(* Logix 5000 project; controller BreakGroup_US vendor 1 type 14 code 211 rev 32.16; software revision 32.05 *)

TASK MainTask (continuous, watchdog 500 ms) : MainProgram
TASK MCP_Panel (periodic, rate 50 ms, priority 10, watchdog 500 ms) : Station_10, Station_20, Station_30, Station_40, Station_50, Station_60, Station_70, Station_80, Gantry_01_Vertical, Gantry_01_Horizontal, Gantry_01_Gripper
TASK RCP_Panel (periodic, rate 50 ms, priority 9, watchdog 500 ms) : Gantry_02_Horizontal, Gantry_02_Vertical, Gantry_02_Gripper, Gantry_02_Tilter, Station_90, Oil_Tank_Lift, Station_100, Station_110, Station_120
TASK SafetyTask (periodic, rate 20 ms, priority 10, watchdog 20 ms, safety) : SafetyProgram

MODULES
   Local : vendor 1 type 14 code 211 (ICP 0, rev 32.16)
      POINT_IO : vendor 1 type 12 code 200 (Ethernet 192.168.1.4, ICP 2, rev 11.1)
           MCP_PT01:1:I.0   // Trolley-1 Locking Cylinder Extended
           MCP_PT01:1:I.1   // Trolley-1 Locking Cylinder Retracted
           MCP_PT01:1:I.2   // Trolley Present Sensor
           MCP_PT01:1:I.3   // Trolley Top Side Product Present Sensors
           MCP_PT01:1:I.4   // Trolley-1 Locking Cylinder Extended
           MCP_PT01:1:I.5   // Trolley-1 Locking Cylinder Retracted
           MCP_PT01:1:I.6   // Trolley Present Sensor
         Servo_RCP : vendor 315 type 14 code 24 (Ethernet 192.168.1.12, rev 1.1, StandardDataDriven RPI 20 ms)
         STN_50_INDEX : vendor 315 type 43 code 25 (Ethernet 192.168.1.30, rev 1.1, StandardDataDriven RPI 20 ms)
         Servo_MCP : vendor 315 type 14 code 24 (Ethernet 192.168.1.11, rev 1.1, StandardDataDriven RPI 20 ms)
         STN_100_INDEX : vendor 315 type 43 code 25 (Ethernet 192.168.1.31, rev 1.1, StandardDataDriven RPI 20 ms)
         STN_110_INDEX : vendor 315 type 43 code 25 (Ethernet 192.168.1.32, rev 1.1, StandardDataDriven RPI 20 ms)
         STN_120_INDEX : vendor 315 type 43 code 25 (Ethernet 192.168.1.33, rev 1.1, StandardDataDriven RPI 20 ms)
         MCP_PT01 : 1734-AENTR (Ethernet 192.168.1.7, rev 7.14, Output RPI 20 ms)
             : 1734-IB8 (PointIO 20, rev 3.1)
             : 1734-IB8 (PointIO 8, rev 3.1)
             : 1734-IB8 (PointIO 7, rev 3.1)
            Slot_01 : 1734-IB8 (PointIO 1, rev 3.1)
             : 1734-IB8 (PointIO 5, rev 3.1)
             : 1734-IB8 (PointIO 18, rev 3.1)
             : 1734-IB8 (PointIO 21, rev 3.1)
             : 1734-IB8 (PointIO 9, rev 3.1)
             : 1734-IB8 (PointIO 10, rev 3.1)
             : 1734-IB8 (PointIO 23, rev 3.1)
             : 1734-IB8 (PointIO 2, rev 3.1)
             : 1734-IB8 (PointIO 16, rev 3.1)
             : 1734-IB8 (PointIO 11, rev 3.1)
             : 1734-IB8 (PointIO 17, rev 3.1)
             : 1734-IB8 (PointIO 14, rev 3.1)
             : 1734-IB8 (PointIO 6, rev 3.1)
             : 1734-IB8 (PointIO 24, rev 3.1)
             : 1734-IB8 (PointIO 19, rev 3.1)
             : 1734-IB8 (PointIO 15, rev 3.1)
             : 1734-IB8 (PointIO 22, rev 3.1)
             : 1734-IB8 (PointIO 13, rev 3.1)
             : 1734-IB8 (PointIO 4, rev 3.1)
             : 1734-IB8 (PointIO 12, rev 3.1)
             : 1734-IB8 (PointIO 3, rev 3.1)
             : 1734-OB8 (PointIO 35, rev 3.1)
             : 1734-OB8 (PointIO 30, rev 3.1)
             : 1734-OB8 (PointIO 25, rev 3.1)
             : 1734-OB8 (PointIO 29, rev 3.1)
             : 1734-OB8 (PointIO 34, rev 3.1)
             : 1734-OB8 (PointIO 32, rev 3.1)
             : 1734-OB8 (PointIO 28, rev 3.1)
             : 1734-OB8 (PointIO 26, rev 3.1)
             : 1734-OB8 (PointIO 33, rev 3.1)
             : 1734-OB8 (PointIO 31, rev 3.1)
             : 1734-OB8 (PointIO 27, rev 3.1)
         RCP_PT01 : 1734-AENTR (Ethernet 192.168.1.9, rev 7.14, Output RPI 20 ms)
             : 1734-IB8 (PointIO 6, rev 3.1)
             : 1734-IB8 (PointIO 3, rev 3.1)
             : 1734-IB8 (PointIO 16, rev 3.1)
             : 1734-IB8 (PointIO 14, rev 3.1)
             : 1734-IB8 (PointIO 10, rev 3.1)
             : 1734-IB8 (PointIO 18, rev 3.1)
             : 1734-IB8 (PointIO 19, rev 3.1)
             : 1734-IB8 (PointIO 13, rev 3.1)
             : 1734-IB8 (PointIO 20, rev 3.1)
             : 1734-IB8 (PointIO 24, rev 3.1)
             : 1734-IB8 (PointIO 15, rev 3.1)
             : 1734-IB8 (PointIO 1, rev 3.1)
             : 1734-IB8 (PointIO 9, rev 3.1)
             : 1734-IB8 (PointIO 21, rev 3.1)
             : 1734-IB8 (PointIO 23, rev 3.1)
             : 1734-IB8 (PointIO 12, rev 3.1)
             : 1734-IB8 (PointIO 2, rev 3.1)
             : 1734-IB8 (PointIO 7, rev 3.1)
             : 1734-IB8 (PointIO 8, rev 3.1)
             : 1734-IB8 (PointIO 17, rev 3.1)
             : 1734-IB8 (PointIO 4, rev 3.1)
             : 1734-IB8 (PointIO 5, rev 3.1)
             : 1734-IB8 (PointIO 11, rev 3.1)
             : 1734-IB8 (PointIO 22, rev 3.1)
             : 1734-OB8 (PointIO 27, rev 3.1)
             : 1734-OB8 (PointIO 30, rev 3.1)
             : 1734-OB8 (PointIO 31, rev 3.1)
             : 1734-OB8 (PointIO 26, rev 3.1)
             : 1734-OB8 (PointIO 25, rev 3.1)
             : 1734-OB8 (PointIO 35, rev 3.1)
             : 1734-OB8 (PointIO 33, rev 3.1)
             : 1734-OB8 (PointIO 28, rev 3.1)
             : 1734-OB8 (PointIO 29, rev 3.1)
             : 1734-OB8 (PointIO 32, rev 3.1)
             : 1734-OB8 (PointIO 34, rev 3.1)
         RCP_PT02 : 1734-AENTR (Ethernet 192.168.1.10, rev 7.14, Output RPI 20 ms)
             : vendor 1 type 115 code 210 (PointIO 10, rev 3.1, Input RPI 80 ms)
             : vendor 1 type 115 code 211 (PointIO 9, rev 3.1, Output RPI 80 ms)
             : 1734-OB8 (PointIO 5, rev 3.1)
             : 1734-OB8 (PointIO 2, rev 3.1)
             : 1734-OB8 (PointIO 8, rev 3.1)
             : 1734-OB8 (PointIO 4, rev 3.1)
             : 1734-OB8 (PointIO 3, rev 3.1)
             : 1734-OB8 (PointIO 7, rev 3.1)
             : 1734-OB8 (PointIO 1, rev 3.1)
             : 1734-OB8 (PointIO 6, rev 3.1)
         MCP_PT02 : 1734-AENTR (Ethernet 192.168.1.8, rev 7.14, Output RPI 20 ms)
             : vendor 1 type 115 code 210 (PointIO 9, rev 3.1, Input RPI 80 ms)
             : 1734-OB8 (PointIO 7, rev 3.1)
             : 1734-OB8 (PointIO 6, rev 3.1)
             : vendor 1 type 115 code 211 (PointIO 8, rev 3.1, Output RPI 80 ms)
             : 1734-OB8 (PointIO 5, rev 3.1)
             : 1734-OB8 (PointIO 2, rev 3.1)
             : 1734-OB8 (PointIO 4, rev 3.1)
             : 1734-OB8 (PointIO 1, rev 3.1)
             : 1734-OB8 (PointIO 3, rev 3.1)
      SERVO : vendor 1 type 12 code 200 (ICP 3, Ethernet 192.168.1.5, rev 11.1)
      ROBOTS : vendor 1 type 12 code 200 (ICP 4, Ethernet 192.168.1.6, rev 11.1)
      @fcc730f7@:Partner : vendor 1 type 14 code 171 (ICP 1, rev 32.16)
END_MODULES

ADD_ON_INSTRUCTION INDEX_Block   (* revision 1.0 *)
VAR_IN_OUT
   PD_INPUT : INT[16]; {required}
   PD_OUTPUT : INT[16]; {required}
   CONNECTION_FAULT : BOOL; {required}
END_VAR
VAR_INPUT
   ENABLE_RAPID_STOP : BOOL; {required}
   ENABLE_APPLICATION_STOP : BOOL; {required}
   START_STOP : BOOL; {required}
   ACTIVATE_INHIBIT : BOOL; {required}
   ACTIVATE_STANDBY : BOOL; {required}
   ACTIVATE_DRIVE_TRAIN_2 : BOOL; {required}
   RESET_ERROR : BOOL; {required}
   SETPOINT_SPEED : INT; {required}
   SETPOINT_DECELERATION : INT; {required}
   SETPOINT_ACCELERATION : INT; {required}
   DIGITAL_OUTPUTS : INT; {required}
END_VAR
VAR_OUTPUT
   COMMUNICATION_OK : BOOL; {access Read Only, required}
   MOVIKIT_HEARTBEAT_STAT : BOOL; {access Read Only, required}
   INVERTER_READY : BOOL; {access Read Only, required}
   STO_INACTIVE : BOOL; {access Read Only, required}
   BRAKE_RELEASED : BOOL; {access Read Only, required}
   OUTPUTSTAGE_ENABLED : BOOL; {access Read Only, required}
   DRIVE_ACTIVE : BOOL; {access Read Only, required}
   WARNING : BOOL; {access Read Only, required}
   ERROR : BOOL; {access Read Only, required}
   DRIVE_TRAIN_2_ACTIVE : BOOL; {access Read Only, required}
   SAFETY_CARD_IN_PLC : BOOL; {access Read Only, required}
   STANDBY_ACTIVE : BOOL; {access Read Only, required}
   VELOCITY_TARGET_ACTUAL_COMPARISON : BOOL; {access Read Only, required}
   ACTUAL_SPEED : INT; {access Read Only, required}
   FAULT_NO : INT; {access Read Only, required}
   ACTUAL_CURRENT : INT; {access Read Only, required}
   DIGITAL_INPUTS : INT; {access Read Only, required}
END_VAR
VAR_INPUT
   RELEASE_BRAKE : BOOL; {access Read Only, required}
   HEART_BEAT_CTRL : BOOL; {access Read Only, required}
   JOG_POS : BOOL; {required}
   JOG_REV : BOOL; {required}
   Rel_ACC : BOOL; {required}
END_VAR
VAR
   L_PDInput : INT[5];
   L_PDOutput : INT[5];
END_VAR

ROUTINE Logic   (* structured text *)
   
   
   if (NOT CONNECTION_FAULT) then
   
   	COMMUNICATION_OK := 1;
   	//Bei fehlerfreiem Lesen werden die Prozesseingangsdaten verarbeitet
       //Zuweisen der einzelnen belegten Ausgänge des Steuerwortes
   	CPS(PD_INPUT[0], L_PDInput[0], 		5);
   
   	//Assigning the StatusBits to the OUTPUT vars of the function block
   
   	//Statusword
   	INVERTER_READY 						:= L_PDInput[0].0;
   	STO_INACTIVE						:= L_PDInput[0].1;
   	OUTPUTSTAGE_ENABLED					:= L_PDInput[0].2;
   	BRAKE_RELEASED						:= L_PDInput[0].3;
   	DRIVE_ACTIVE 						:= L_PDInput[0].4;
   //	N.N. 							:= L_PDInput[0].5;
   //	N.N.							:= L_PDInput[0].6;
   //	N.N.								:= L_PDInput[0].7;
   	ERROR 								:= L_PDInput[0].8;
   	WARNING								:= L_PDInput[0].9;
   	DRIVE_TRAIN_2_ACTIVE 				:= L_PDInput[0].10;
   	VELOCITY_TARGET_ACTUAL_COMPARISON 	:= L_PDInput[0].11;
   //	N.N.								:= L_PDInput[0].12;
   	SAFETY_CARD_IN_PLC					:= L_PDInput[0].13;
   	STANDBY_ACTIVE						:= L_PDInput[0].14;
   	MOVIKIT_HEARTBEAT_STAT				:= L_PDInput[0].15;
   
   	//Assigning the actual values to the OUTPUTS of the function block
   	ACTUAL_SPEED 						:= L_PDInput[1];
   	FAULT_NO 							:= L_PDInput[2];
   	ACTUAL_CURRENT 						:= L_PDInput[3];
   	DIGITAL_INPUTS 						:= L_PDInput[4];
   
   
   	//=================================================================================================
   	//=================================================================================================
   
   	//Assigning the Bits of the function block INPUTS to the Local Controlword
   	L_PDOutput[0].0						:= ENABLE_RAPID_STOP;
   	L_PDOutput[0].1 					:= ENABLE_APPLICATION_STOP;
   	L_PDOutput[0].3 					:= RELEASE_BRAKE;
   	L_PDOutput[0].7						:= START_STOP;
   	L_PDOutput[0].8 					:= RESET_ERROR;
   	L_PDOutput[0].10					:= ACTIVATE_DRIVE_TRAIN_2;
   	L_PDOutput[0].13					:= ACTIVATE_INHIBIT;
   	L_PDOutput[0].14					:= ACTIVATE_STANDBY;
   	L_PDOutput[0].15 					:= HEART_BEAT_CTRL;
   	//Setting the remaining bits on inactive
   	L_PDOutput[0].2 					:= 0;
   	L_PDOutput[0].4 					:= JOG_POS;
   	L_PDOutput[0].5 					:= JOG_REV;
   	L_PDOutput[0].6 					:= Rel_ACC;
   	L_PDOutput[0].9 					:= 0;
   	L_PDOutput[0].11 					:= 0;
   	L_PDOutput[0].12					:= 0;
   
   
   
   	//Setting the INPUTS of the function block to Local Variables for Outputs
   	L_PDOutput[1] 						:= SETPOINT_SPEED;
   	L_PDOutput[2]						:= SETPOINT_ACCELERATION;
   	L_PDOutput[3]						:= SETPOINT_DECELERATION;
   	L_PDOutput[4]						:= DIGITAL_OUTPUTS;
   
   
   else
   	COMMUNICATION_OK := 0;
   	//Delete the local vars for OUTPUTS in case of comm error
   	L_PDOutput[0].0						:= 0;
   	L_PDOutput[0].1 					:= 0;
   	L_PDOutput[0].3 					:= 0;
   	L_PDOutput[0].7						:= 0;
   	L_PDOutput[0].8 					:= 0;
   	L_PDOutput[0].10					:= 0;
   	L_PDOutput[0].12					:= 0;
   	L_PDOutput[0].13					:= 0;
   	L_PDOutput[0].14					:= 0;
   	L_PDOutput[0].2 					:= 0;
   	L_PDOutput[0].4 					:= 0;
   	L_PDOutput[0].5 					:= 0;
   	L_PDOutput[0].6 					:= 0;
   	L_PDOutput[0].9 					:= 0;
   	L_PDOutput[0].11 					:= 0;
   	L_PDOutput[0].15 					:= 0; //Heratbeat?
   
   	L_PDOutput[1] 					:= 0;
   	L_PDOutput[2]				:= 0;
   	L_PDOutput[3]				:= 0;
   	L_PDOutput[4]						:= 0;
   end_IF;
   
   
   CPS(L_PDOutput[0], PD_OUTPUT[0], 10);
   
END_ROUTINE
END_ADD_ON_INSTRUCTION

ADD_ON_INSTRUCTION MCP_Servo_01   (* revision 1.0, vendor SEW *)
VAR_INPUT
   Start_Offest_Num : SINT; {required}
END_VAR
VAR_IN_OUT
   SEW_DataType_In : INT[48]; {required}
   SEW_DataType_Out : INT[48]; {required}
END_VAR
VAR_OUTPUT
   Inverter_Ready : BOOL; {access Read Only, visible}
   STO_InActive : BOOL; {visible}
   PwR_Stge_oN : BOOL; {visible}
   Brake_Released : BOOL; {visible}
   Motor_Turning : BOOL; {visible}
   Referenced_Drive : BOOL; {visible}
   NewRelativePosition_Applied : BOOL; {visible}
   InPosition : BOOL; {visible}
   Fault_Active : BOOL; {visible}
   Warning_Active : BOOL; {visible}
   SpdSetPoint_Reached : BOOL; {visible}
   SftWreLiMits_DisAble : BOOL; {visible}
   FCBaCtive : BOOL; {visible}
   StandByMode_Active : BOOL; {visible}
   MoviKitHandshakeBit_Out : BOOL; {visible}
   Actual_Speed : REAL; {visible}
   Fault_Num : SINT; {visible}   // High word fault or inverter status
   Status_Suberror_Num : SINT; {visible}   // Low word fault sub error number
   Actual_MtrTorque : REAL; {visible}
   Digital_Inputs : INT; {visible}
   Actual_Mode : INT; {visible}
   Actual_Pos : REAL; {visible}
END_VAR
VAR_INPUT
   Enable_EsTop : BOOL := 1; {visible}
   Enable_Stop : BOOL; {required}
   Release_Brake : BOOL; {visible}
   Jog_Pos : BOOL; {visible}
   Jog_Neg : BOOL; {visible}
   Accept_Rel_Position : BOOL; {visible}
   Start_Stop : BOOL; {required}
   Fault_Reset : BOOL; {required}
   DisAbleSW_Limits : BOOL; {visible}
   Inverter_Inhibit : BOOL; {visible}
   StandByMode_Enable : BOOL; {visible}
   MoviKitHandShakeBit_In : BOOL; {visible}
   Speed : REAL; {required}
   Accel_Ramp : REAL; {required}
   Decel_Ramp : REAL; {required}
   Digital_Outputs : INT; {visible}
   Application_Mode : INT; {required}
   Target_Position : REAL; {required}
   PositionDecimal_Place : SINT; {visible}
   SpeedDecimal_PLace : SINT; {visible}
   Accel_DecelDecimal_Place : SINT; {visible}
   Controller_Disconnected : BOOL; {required}
END_VAR
VAR
   L_PD_OUT : INT[8]; {access None}
   L_PD_IN : INT[8]; {access None}
   L_Position_OUT : DINT; {access None}
   L_Position_In : DINT; {access None}
END_VAR

ROUTINE Logic   (* ladder *)
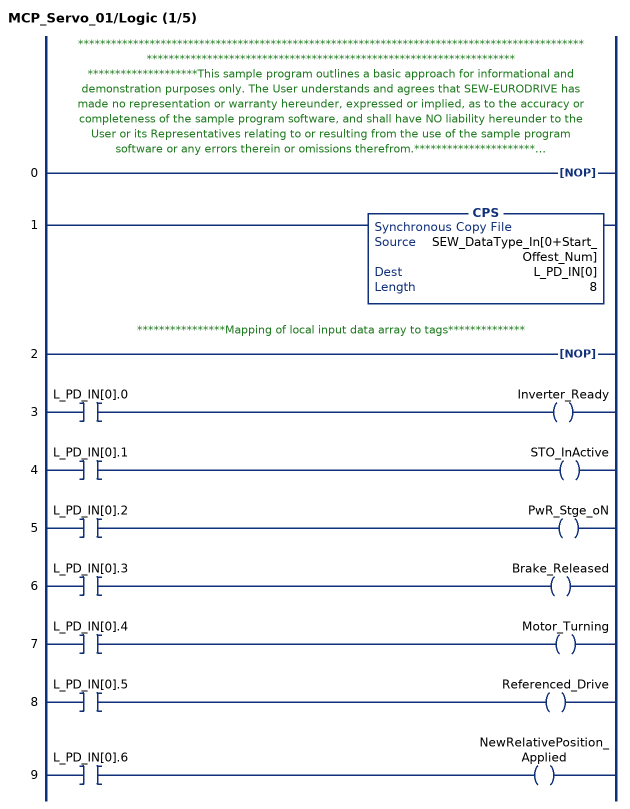
   // ***************************************************************************************************************************************************************
   // ********************This sample program outlines a basic approach for informational and demonstration purposes only. The User understands and agrees that SEW-EURODRIVE has made no representation or warranty hereunder, expressed or implied, as to the accuracy or completeness of the sample program software, and shall have NO liability hereunder to the User or its Representatives relating to or resulting from the use of the sample program software or any errors therein or omissions therefrom.***********************
   // **********************************************************************************************************************************************************
   0: NOP();
   1: CPS(SEW_DataType_In[0+Start_Offest_Num],L_PD_IN[0],8);
   // ****************Mapping of local input data array to tags**************
   2: NOP();
   3: XIC(L_PD_IN[0].0)OTE(Inverter_Ready);
   4: XIC(L_PD_IN[0].1)OTE(STO_InActive);
   5: XIC(L_PD_IN[0].2)OTE(PwR_Stge_oN);
   6: XIC(L_PD_IN[0].3)OTE(Brake_Released);
   7: XIC(L_PD_IN[0].4)OTE(Motor_Turning);
   8: XIC(L_PD_IN[0].5)OTE(Referenced_Drive);
   9: XIC(L_PD_IN[0].6)OTE(NewRelativePosition_Applied);
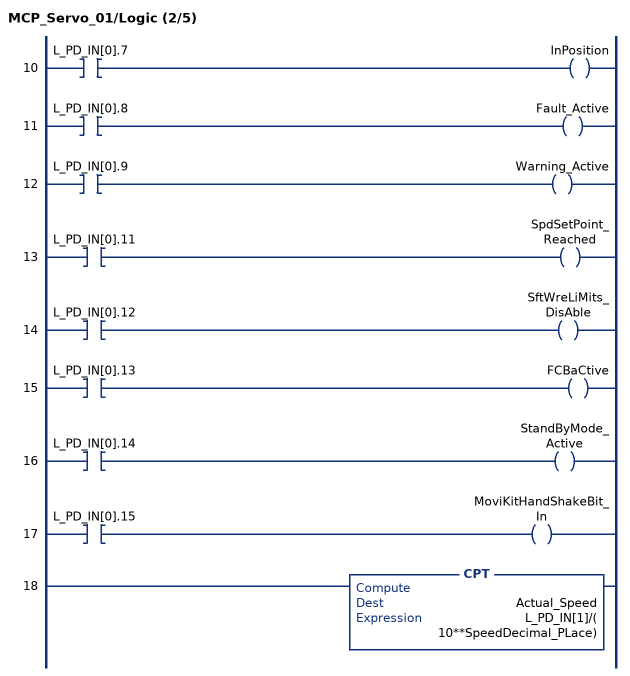
   10: XIC(L_PD_IN[0].7)OTE(InPosition);
   11: XIC(L_PD_IN[0].8)OTE(Fault_Active);
   12: XIC(L_PD_IN[0].9)OTE(Warning_Active);
   13: XIC(L_PD_IN[0].11)OTE(SpdSetPoint_Reached);
   14: XIC(L_PD_IN[0].12)OTE(SftWreLiMits_DisAble);
   15: XIC(L_PD_IN[0].13)OTE(FCBaCtive);
   16: XIC(L_PD_IN[0].14)OTE(StandByMode_Active);
   17: XIC(L_PD_IN[0].15)OTE(MoviKitHandShakeBit_In);
   18: CPT(Actual_Speed,L_PD_IN[1]/(10**SpeedDecimal_PLace));
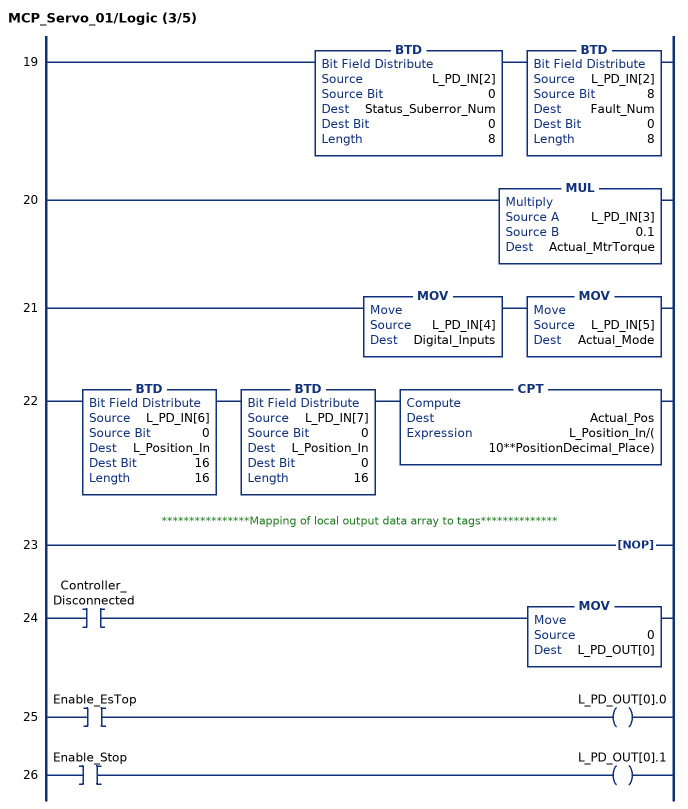
   19: BTD(L_PD_IN[2],0,Status_Suberror_Num,0,8)BTD(L_PD_IN[2],8,Fault_Num,0,8);
   20: MUL(L_PD_IN[3],0.1,Actual_MtrTorque);
   21: MOV(L_PD_IN[4],Digital_Inputs)MOV(L_PD_IN[5],Actual_Mode);
   22: BTD(L_PD_IN[6],0,L_Position_In,16,16)BTD(L_PD_IN[7],0,L_Position_In,0,16)CPT(Actual_Pos,L_Position_In/(10**PositionDecimal_Place));
   // ****************Mapping of local output data array to tags**************
   23: NOP();
   24: XIC(Controller_Disconnected)MOV(0,L_PD_OUT[0]);
   25: XIC(Enable_EsTop)OTE(L_PD_OUT[0].0);
   26: XIC(Enable_Stop)OTE(L_PD_OUT[0].1);
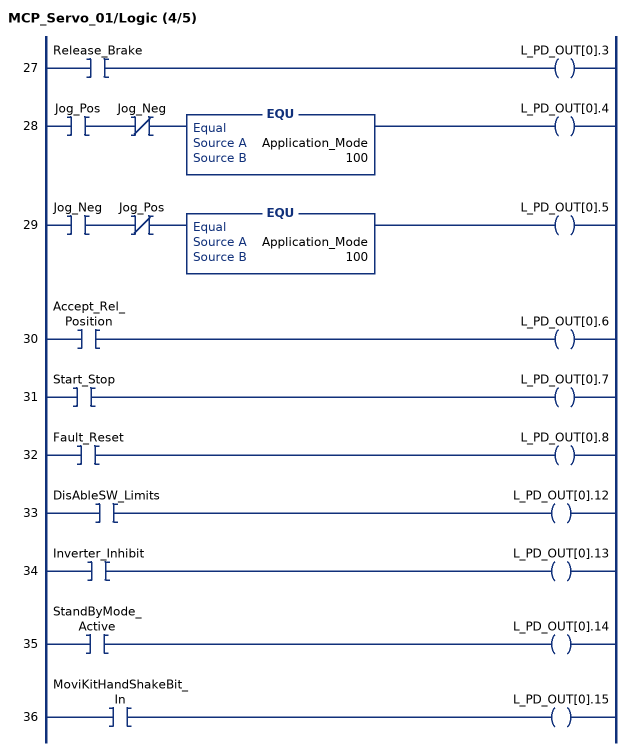
   27: XIC(Release_Brake)OTE(L_PD_OUT[0].3);
   28: XIC(Jog_Pos)XIO(Jog_Neg)EQU(Application_Mode,100)OTE(L_PD_OUT[0].4);
   29: XIC(Jog_Neg)XIO(Jog_Pos)EQU(Application_Mode,100)OTE(L_PD_OUT[0].5);
   30: XIC(Accept_Rel_Position)OTE(L_PD_OUT[0].6);
   31: XIC(Start_Stop)OTE(L_PD_OUT[0].7);
   32: XIC(Fault_Reset)OTE(L_PD_OUT[0].8);
   33: XIC(DisAbleSW_Limits)OTE(L_PD_OUT[0].12);
   34: XIC(Inverter_Inhibit)OTE(L_PD_OUT[0].13);
   35: XIC(StandByMode_Active)OTE(L_PD_OUT[0].14);
   36: XIC(MoviKitHandShakeBit_In)OTE(L_PD_OUT[0].15);
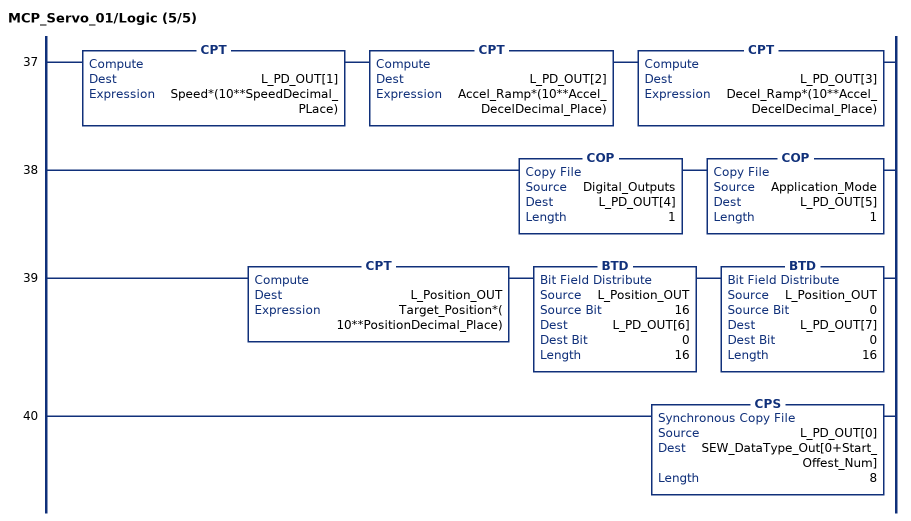
   37: CPT(L_PD_OUT[1],Speed*(10**SpeedDecimal_PLace))CPT(L_PD_OUT[2],Accel_Ramp*(10**Accel_DecelDecimal_Place))CPT(L_PD_OUT[3],Decel_Ramp*(10**Accel_DecelDecimal_Place));
   38: COP(Digital_Outputs,L_PD_OUT[4],1)COP(Application_Mode,L_PD_OUT[5],1);
   39: CPT(L_Position_OUT,Target_Position*(10**PositionDecimal_Place))BTD(L_Position_OUT,16,L_PD_OUT[6],0,16)BTD(L_Position_OUT,0,L_PD_OUT[7],0,16);
   40: CPS(L_PD_OUT[0],SEW_DataType_Out[0+Start_Offest_Num],8);
END_ROUTINE
END_ADD_ON_INSTRUCTION

ADD_ON_INSTRUCTION MCP_Servo_02   (* revision 1.0, vendor SEW *)
VAR_INPUT
   Start_Offest_Num : SINT; {required}
END_VAR
VAR_IN_OUT
   SEW_DataType_In : INT[248]; {required}
   SEW_DataType_Out : INT[248]; {required}
END_VAR
VAR_OUTPUT
   Inverter_Ready : BOOL; {access Read Only, visible}
   STO_InActive : BOOL; {visible}
   PwR_Stge_oN : BOOL; {visible}
   Brake_Released : BOOL; {visible}
   Motor_Turning : BOOL; {visible}
   Referenced_Drive : BOOL; {visible}
   NewRelativePosition_Applied : BOOL; {visible}
   InPosition : BOOL; {visible}
   Fault_Active : BOOL; {visible}
   Warning_Active : BOOL; {visible}
   SpdSetPoint_Reached : BOOL; {visible}
   SftWreLiMits_DisAble : BOOL; {visible}
   FCBaCtive : BOOL; {visible}
   StandByMode_Active : BOOL; {visible}
   MoviKitHandshakeBit_Out : BOOL; {visible}
   Actual_Speed : REAL; {visible}
   Fault_Num : SINT; {visible}   // High word fault or inverter status
   Status_Suberror_Num : SINT; {visible}   // Low word fault sub error number
   Actual_MtrTorque : REAL; {visible}
   Digital_Inputs : INT; {visible}
   Actual_Mode : INT; {visible}
   Actual_Pos : REAL; {visible}
END_VAR
VAR_INPUT
   Enable_EsTop : BOOL := 1; {visible}
   Enable_Stop : BOOL; {required}
   Release_Brake : BOOL; {visible}
   Jog_Pos : BOOL; {visible}
   Jog_Neg : BOOL; {visible}
   Accept_Rel_Position : BOOL; {visible}
   Start_Stop : BOOL; {required}
   Fault_Reset : BOOL; {required}
   DisAbleSW_Limits : BOOL; {visible}
   Inverter_Inhibit : BOOL; {visible}
   StandByMode_Enable : BOOL; {visible}
   MoviKitHandShakeBit_In : BOOL; {visible}
   Speed : REAL; {required}
   Accel_Ramp : REAL; {required}
   Decel_Ramp : REAL; {required}
   Digital_Outputs : INT; {visible}
   Application_Mode : INT; {required}
   Target_Position : REAL; {required}
   PositionDecimal_Place : SINT; {visible}
   SpeedDecimal_PLace : SINT; {visible}
   Accel_DecelDecimal_Place : SINT; {visible}
   Controller_Disconnected : BOOL; {required}
END_VAR
VAR
   L_PD_OUT : INT[8]; {access None}
   L_PD_IN : INT[8]; {access None}
   L_Position_OUT : DINT; {access None}
   L_Position_In : DINT; {access None}
END_VAR

ROUTINE Logic   (* ladder *)
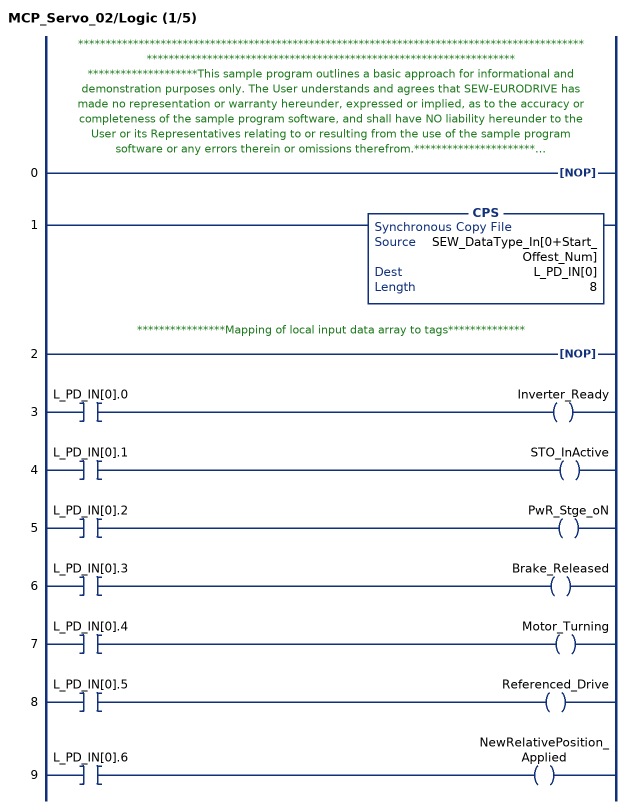
   // ***************************************************************************************************************************************************************
   // ********************This sample program outlines a basic approach for informational and demonstration purposes only. The User understands and agrees that SEW-EURODRIVE has made no representation or warranty hereunder, expressed or implied, as to the accuracy or completeness of the sample program software, and shall have NO liability hereunder to the User or its Representatives relating to or resulting from the use of the sample program software or any errors therein or omissions therefrom.***********************
   // **********************************************************************************************************************************************************
   0: NOP();
   1: CPS(SEW_DataType_In[0+Start_Offest_Num],L_PD_IN[0],8);
   // ****************Mapping of local input data array to tags**************
   2: NOP();
   3: XIC(L_PD_IN[0].0)OTE(Inverter_Ready);
   4: XIC(L_PD_IN[0].1)OTE(STO_InActive);
   5: XIC(L_PD_IN[0].2)OTE(PwR_Stge_oN);
   6: XIC(L_PD_IN[0].3)OTE(Brake_Released);
   7: XIC(L_PD_IN[0].4)OTE(Motor_Turning);
   8: XIC(L_PD_IN[0].5)OTE(Referenced_Drive);
   9: XIC(L_PD_IN[0].6)OTE(NewRelativePosition_Applied);
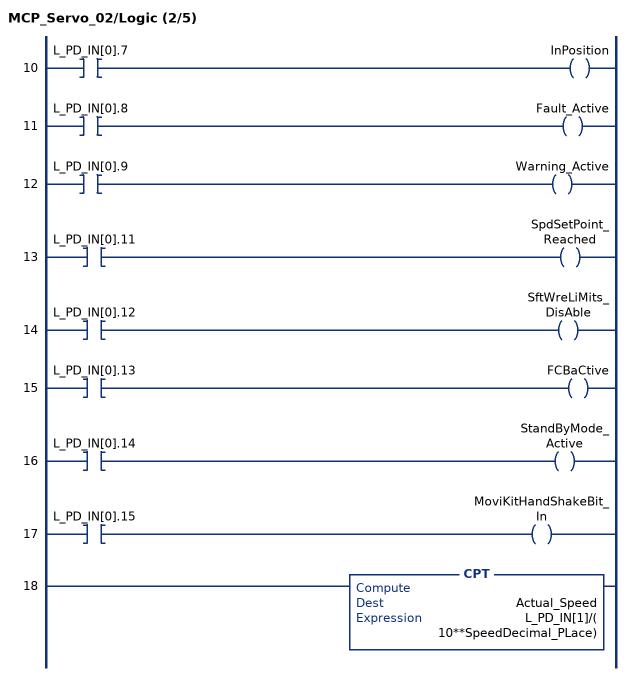
   10: XIC(L_PD_IN[0].7)OTE(InPosition);
   11: XIC(L_PD_IN[0].8)OTE(Fault_Active);
   12: XIC(L_PD_IN[0].9)OTE(Warning_Active);
   13: XIC(L_PD_IN[0].11)OTE(SpdSetPoint_Reached);
   14: XIC(L_PD_IN[0].12)OTE(SftWreLiMits_DisAble);
   15: XIC(L_PD_IN[0].13)OTE(FCBaCtive);
   16: XIC(L_PD_IN[0].14)OTE(StandByMode_Active);
   17: XIC(L_PD_IN[0].15)OTE(MoviKitHandShakeBit_In);
   18: CPT(Actual_Speed,L_PD_IN[1]/(10**SpeedDecimal_PLace));
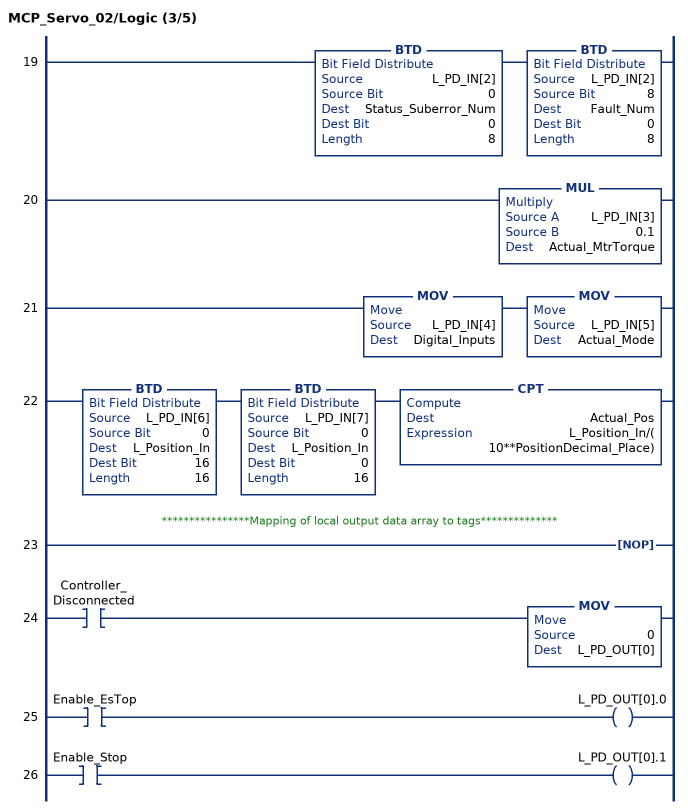
   19: BTD(L_PD_IN[2],0,Status_Suberror_Num,0,8)BTD(L_PD_IN[2],8,Fault_Num,0,8);
   20: MUL(L_PD_IN[3],0.1,Actual_MtrTorque);
   21: MOV(L_PD_IN[4],Digital_Inputs)MOV(L_PD_IN[5],Actual_Mode);
   22: BTD(L_PD_IN[6],0,L_Position_In,16,16)BTD(L_PD_IN[7],0,L_Position_In,0,16)CPT(Actual_Pos,L_Position_In/(10**PositionDecimal_Place));
   // ****************Mapping of local output data array to tags**************
   23: NOP();
   24: XIC(Controller_Disconnected)MOV(0,L_PD_OUT[0]);
   25: XIC(Enable_EsTop)OTE(L_PD_OUT[0].0);
   26: XIC(Enable_Stop)OTE(L_PD_OUT[0].1);
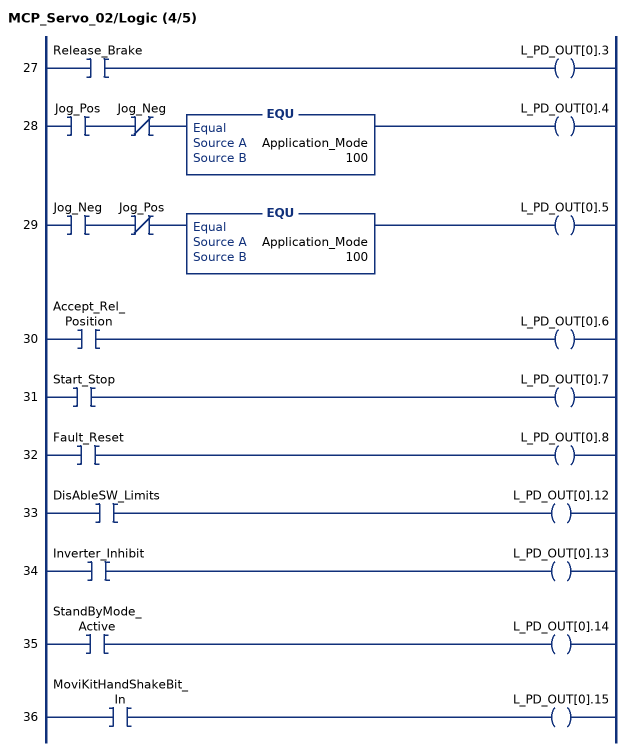
   27: XIC(Release_Brake)OTE(L_PD_OUT[0].3);
   28: XIC(Jog_Pos)XIO(Jog_Neg)EQU(Application_Mode,100)OTE(L_PD_OUT[0].4);
   29: XIC(Jog_Neg)XIO(Jog_Pos)EQU(Application_Mode,100)OTE(L_PD_OUT[0].5);
   30: XIC(Accept_Rel_Position)OTE(L_PD_OUT[0].6);
   31: XIC(Start_Stop)OTE(L_PD_OUT[0].7);
   32: XIC(Fault_Reset)OTE(L_PD_OUT[0].8);
   33: XIC(DisAbleSW_Limits)OTE(L_PD_OUT[0].12);
   34: XIC(Inverter_Inhibit)OTE(L_PD_OUT[0].13);
   35: XIC(StandByMode_Active)OTE(L_PD_OUT[0].14);
   36: XIC(MoviKitHandShakeBit_In)OTE(L_PD_OUT[0].15);
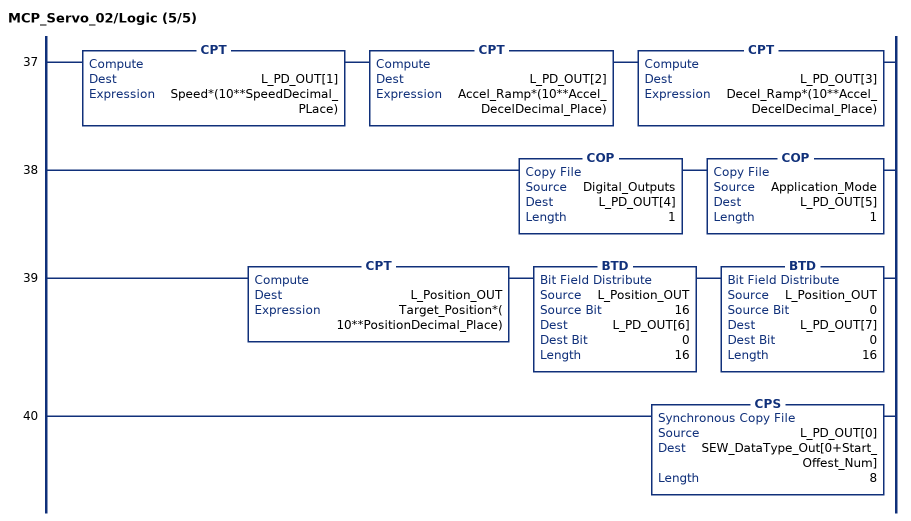
   37: CPT(L_PD_OUT[1],Speed*(10**SpeedDecimal_PLace))CPT(L_PD_OUT[2],Accel_Ramp*(10**Accel_DecelDecimal_Place))CPT(L_PD_OUT[3],Decel_Ramp*(10**Accel_DecelDecimal_Place));
   38: COP(Digital_Outputs,L_PD_OUT[4],1)COP(Application_Mode,L_PD_OUT[5],1);
   39: CPT(L_Position_OUT,Target_Position*(10**PositionDecimal_Place))BTD(L_Position_OUT,16,L_PD_OUT[6],0,16)BTD(L_Position_OUT,0,L_PD_OUT[7],0,16);
   40: CPS(L_PD_OUT[0],SEW_DataType_Out[0+Start_Offest_Num],8);
END_ROUTINE
END_ADD_ON_INSTRUCTION

ADD_ON_INSTRUCTION RCP_Servo_01   (* revision 1.0, vendor SEW *)
VAR_INPUT
   Start_Offest_Num : SINT; {required}
END_VAR
VAR_IN_OUT
   SEW_DataType_In : INT[48]; {required}
   SEW_DataType_Out : INT[48]; {required}
END_VAR
VAR_OUTPUT
   Inverter_Ready : BOOL; {access Read Only, visible}
   STO_InActive : BOOL; {visible}
   PwR_Stge_oN : BOOL; {visible}
   Brake_Released : BOOL; {visible}
   Motor_Turning : BOOL; {visible}
   Referenced_Drive : BOOL; {visible}
   NewRelativePosition_Applied : BOOL; {visible}
   InPosition : BOOL; {visible}
   Fault_Active : BOOL; {visible}
   Warning_Active : BOOL; {visible}
   SpdSetPoint_Reached : BOOL; {visible}
   SftWreLiMits_DisAble : BOOL; {visible}
   FCBaCtive : BOOL; {visible}
   StandByMode_Active : BOOL; {visible}
   MoviKitHandshakeBit_Out : BOOL; {visible}
   Actual_Speed : REAL; {visible}
   Fault_Num : SINT; {visible}   // High word fault or inverter status
   Status_Suberror_Num : SINT; {visible}   // Low word fault sub error number
   Actual_MtrTorque : REAL; {visible}
   Digital_Inputs : INT; {visible}
   Actual_Mode : INT; {visible}
   Actual_Pos : REAL; {visible}
END_VAR
VAR_INPUT
   Enable_EsTop : BOOL := 1; {visible}
   Enable_Stop : BOOL; {required}
   Release_Brake : BOOL; {visible}
   Jog_Pos : BOOL; {visible}
   Jog_Neg : BOOL; {visible}
   Accept_Rel_Position : BOOL; {visible}
   Start_Stop : BOOL; {required}
   Fault_Reset : BOOL; {required}
   DisAbleSW_Limits : BOOL; {visible}
   Inverter_Inhibit : BOOL; {visible}
   StandByMode_Enable : BOOL; {visible}
   MoviKitHandShakeBit_In : BOOL; {visible}
   Speed : REAL; {required}
   Accel_Ramp : REAL; {required}
   Decel_Ramp : REAL; {required}
   Digital_Outputs : INT; {visible}
   Application_Mode : INT; {required}
   Target_Position : REAL; {required}
   PositionDecimal_Place : SINT; {visible}
   SpeedDecimal_PLace : SINT; {visible}
   Accel_DecelDecimal_Place : SINT; {visible}
   Controller_Disconnected : BOOL; {required}
END_VAR
VAR
   L_PD_OUT : INT[8]; {access None}
   L_PD_IN : INT[8]; {access None}
   L_Position_OUT : DINT; {access None}
   L_Position_In : DINT; {access None}
END_VAR

ROUTINE Logic   (* ladder *)
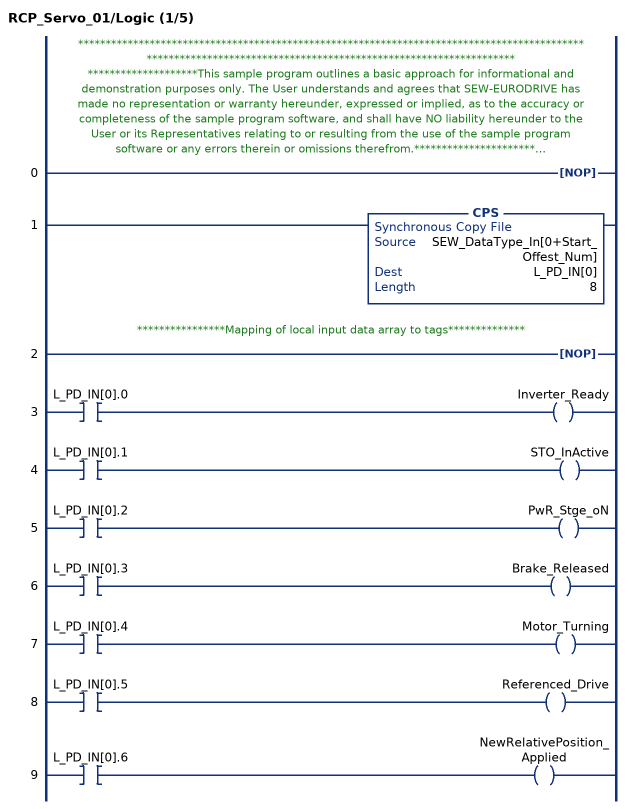
   // ***************************************************************************************************************************************************************
   // ********************This sample program outlines a basic approach for informational and demonstration purposes only. The User understands and agrees that SEW-EURODRIVE has made no representation or warranty hereunder, expressed or implied, as to the accuracy or completeness of the sample program software, and shall have NO liability hereunder to the User or its Representatives relating to or resulting from the use of the sample program software or any errors therein or omissions therefrom.***********************
   // **********************************************************************************************************************************************************
   0: NOP();
   1: CPS(SEW_DataType_In[0+Start_Offest_Num],L_PD_IN[0],8);
   // ****************Mapping of local input data array to tags**************
   2: NOP();
   3: XIC(L_PD_IN[0].0)OTE(Inverter_Ready);
   4: XIC(L_PD_IN[0].1)OTE(STO_InActive);
   5: XIC(L_PD_IN[0].2)OTE(PwR_Stge_oN);
   6: XIC(L_PD_IN[0].3)OTE(Brake_Released);
   7: XIC(L_PD_IN[0].4)OTE(Motor_Turning);
   8: XIC(L_PD_IN[0].5)OTE(Referenced_Drive);
   9: XIC(L_PD_IN[0].6)OTE(NewRelativePosition_Applied);
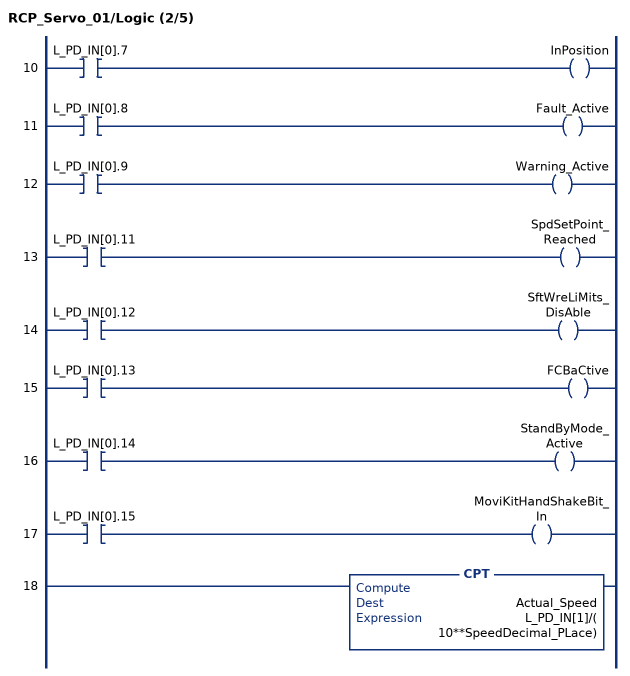
   10: XIC(L_PD_IN[0].7)OTE(InPosition);
   11: XIC(L_PD_IN[0].8)OTE(Fault_Active);
   12: XIC(L_PD_IN[0].9)OTE(Warning_Active);
   13: XIC(L_PD_IN[0].11)OTE(SpdSetPoint_Reached);
   14: XIC(L_PD_IN[0].12)OTE(SftWreLiMits_DisAble);
   15: XIC(L_PD_IN[0].13)OTE(FCBaCtive);
   16: XIC(L_PD_IN[0].14)OTE(StandByMode_Active);
   17: XIC(L_PD_IN[0].15)OTE(MoviKitHandShakeBit_In);
   18: CPT(Actual_Speed,L_PD_IN[1]/(10**SpeedDecimal_PLace));
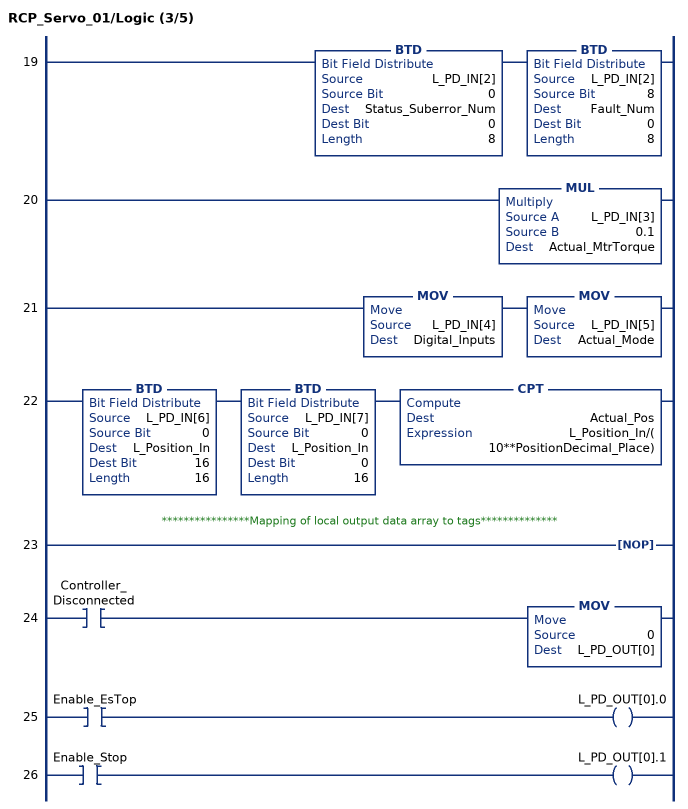
   19: BTD(L_PD_IN[2],0,Status_Suberror_Num,0,8)BTD(L_PD_IN[2],8,Fault_Num,0,8);
   20: MUL(L_PD_IN[3],0.1,Actual_MtrTorque);
   21: MOV(L_PD_IN[4],Digital_Inputs)MOV(L_PD_IN[5],Actual_Mode);
   22: BTD(L_PD_IN[6],0,L_Position_In,16,16)BTD(L_PD_IN[7],0,L_Position_In,0,16)CPT(Actual_Pos,L_Position_In/(10**PositionDecimal_Place));
   // ****************Mapping of local output data array to tags**************
   23: NOP();
   24: XIC(Controller_Disconnected)MOV(0,L_PD_OUT[0]);
   25: XIC(Enable_EsTop)OTE(L_PD_OUT[0].0);
   26: XIC(Enable_Stop)OTE(L_PD_OUT[0].1);
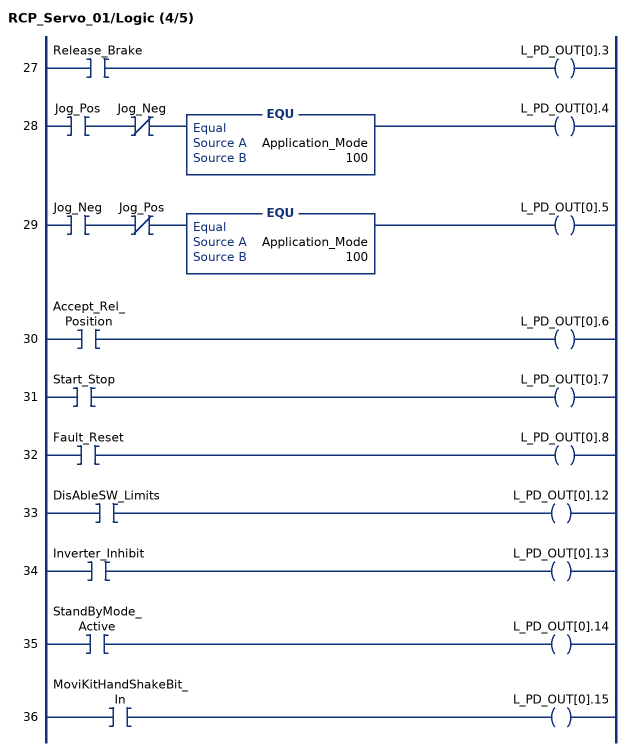
   27: XIC(Release_Brake)OTE(L_PD_OUT[0].3);
   28: XIC(Jog_Pos)XIO(Jog_Neg)EQU(Application_Mode,100)OTE(L_PD_OUT[0].4);
   29: XIC(Jog_Neg)XIO(Jog_Pos)EQU(Application_Mode,100)OTE(L_PD_OUT[0].5);
   30: XIC(Accept_Rel_Position)OTE(L_PD_OUT[0].6);
   31: XIC(Start_Stop)OTE(L_PD_OUT[0].7);
   32: XIC(Fault_Reset)OTE(L_PD_OUT[0].8);
   33: XIC(DisAbleSW_Limits)OTE(L_PD_OUT[0].12);
   34: XIC(Inverter_Inhibit)OTE(L_PD_OUT[0].13);
   35: XIC(StandByMode_Active)OTE(L_PD_OUT[0].14);
   36: XIC(MoviKitHandShakeBit_In)OTE(L_PD_OUT[0].15);
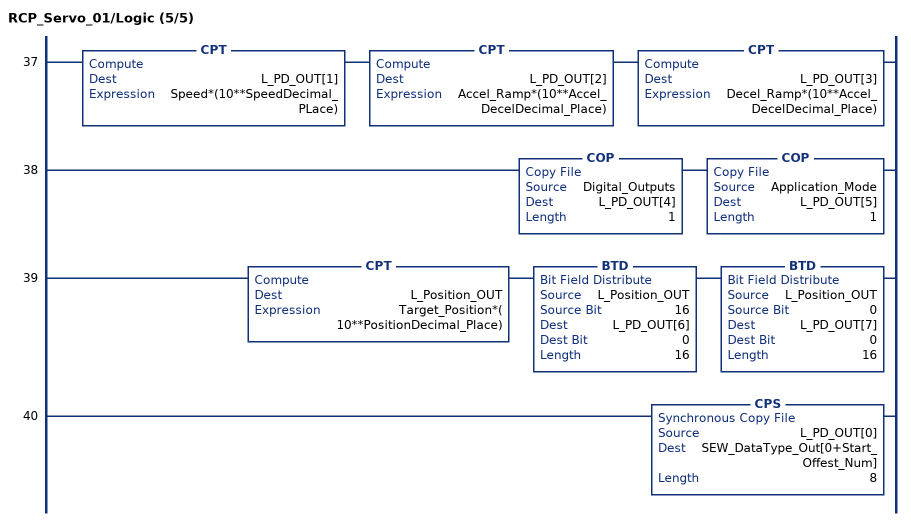
   37: CPT(L_PD_OUT[1],Speed*(10**SpeedDecimal_PLace))CPT(L_PD_OUT[2],Accel_Ramp*(10**Accel_DecelDecimal_Place))CPT(L_PD_OUT[3],Decel_Ramp*(10**Accel_DecelDecimal_Place));
   38: COP(Digital_Outputs,L_PD_OUT[4],1)COP(Application_Mode,L_PD_OUT[5],1);
   39: CPT(L_Position_OUT,Target_Position*(10**PositionDecimal_Place))BTD(L_Position_OUT,16,L_PD_OUT[6],0,16)BTD(L_Position_OUT,0,L_PD_OUT[7],0,16);
   40: CPS(L_PD_OUT[0],SEW_DataType_Out[0+Start_Offest_Num],8);
END_ROUTINE
END_ADD_ON_INSTRUCTION

ADD_ON_INSTRUCTION RCP_Servo_02   (* revision 1.0, vendor SEW *)
VAR_INPUT
   Start_Offest_Num : SINT; {required}
END_VAR
VAR_IN_OUT
   SEW_DataType_In : INT[248]; {required}
   SEW_DataType_Out : INT[248]; {required}
END_VAR
VAR_OUTPUT
   Inverter_Ready : BOOL; {access Read Only, visible}
   STO_InActive : BOOL; {visible}
   PwR_Stge_oN : BOOL; {visible}
   Brake_Released : BOOL; {visible}
   Motor_Turning : BOOL; {visible}
   Referenced_Drive : BOOL; {visible}
   NewRelativePosition_Applied : BOOL; {visible}
   InPosition : BOOL; {visible}
   Fault_Active : BOOL; {visible}
   Warning_Active : BOOL; {visible}
   SpdSetPoint_Reached : BOOL; {visible}
   SftWreLiMits_DisAble : BOOL; {visible}
   FCBaCtive : BOOL; {visible}
   StandByMode_Active : BOOL; {visible}
   MoviKitHandshakeBit_Out : BOOL; {visible}
   Actual_Speed : REAL; {visible}
   Fault_Num : SINT; {visible}   // High word fault or inverter status
   Status_Suberror_Num : SINT; {visible}   // Low word fault sub error number
   Actual_MtrTorque : REAL; {visible}
   Digital_Inputs : INT; {visible}
   Actual_Mode : INT; {visible}
   Actual_Pos : REAL; {visible}
END_VAR
VAR_INPUT
   Enable_EsTop : BOOL := 1; {visible}
   Enable_Stop : BOOL; {required}
   Release_Brake : BOOL; {visible}
   Jog_Pos : BOOL; {visible}
   Jog_Neg : BOOL; {visible}
   Accept_Rel_Position : BOOL; {visible}
   Start_Stop : BOOL; {required}
   Fault_Reset : BOOL; {required}
   DisAbleSW_Limits : BOOL; {visible}
   Inverter_Inhibit : BOOL; {visible}
   StandByMode_Enable : BOOL; {visible}
   MoviKitHandShakeBit_In : BOOL; {visible}
   Speed : REAL; {required}
   Accel_Ramp : REAL; {required}
   Decel_Ramp : REAL; {required}
   Digital_Outputs : INT; {visible}
   Application_Mode : INT; {required}
   Target_Position : REAL; {required}
   PositionDecimal_Place : SINT; {visible}
   SpeedDecimal_PLace : SINT; {visible}
   Accel_DecelDecimal_Place : SINT; {visible}
   Controller_Disconnected : BOOL; {required}
END_VAR
VAR
   L_PD_OUT : INT[8]; {access None}
   L_PD_IN : INT[8]; {access None}
   L_Position_OUT : DINT; {access None}
   L_Position_In : DINT; {access None}
END_VAR

ROUTINE Logic   (* ladder *)
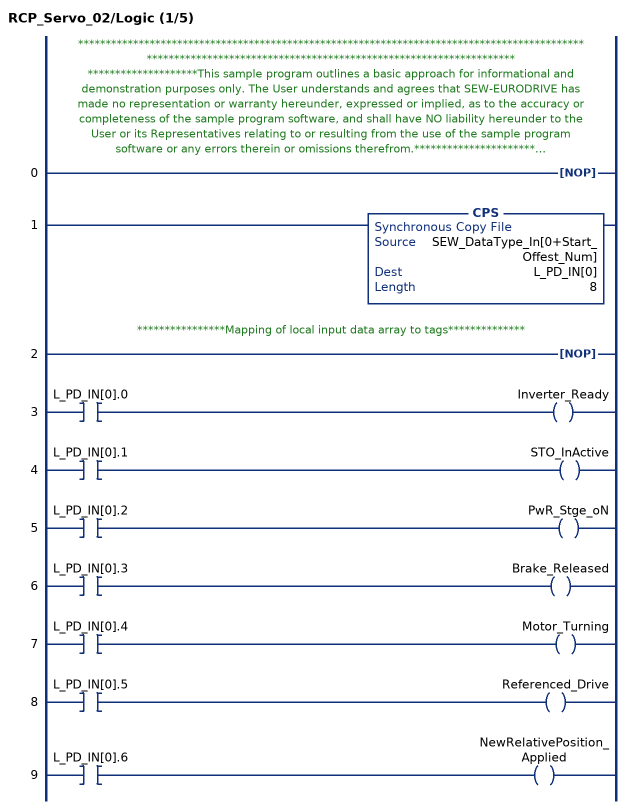
   // ***************************************************************************************************************************************************************
   // ********************This sample program outlines a basic approach for informational and demonstration purposes only. The User understands and agrees that SEW-EURODRIVE has made no representation or warranty hereunder, expressed or implied, as to the accuracy or completeness of the sample program software, and shall have NO liability hereunder to the User or its Representatives relating to or resulting from the use of the sample program software or any errors therein or omissions therefrom.***********************
   // **********************************************************************************************************************************************************
   0: NOP();
   1: CPS(SEW_DataType_In[0+Start_Offest_Num],L_PD_IN[0],8);
   // ****************Mapping of local input data array to tags**************
   2: NOP();
   3: XIC(L_PD_IN[0].0)OTE(Inverter_Ready);
   4: XIC(L_PD_IN[0].1)OTE(STO_InActive);
   5: XIC(L_PD_IN[0].2)OTE(PwR_Stge_oN);
   6: XIC(L_PD_IN[0].3)OTE(Brake_Released);
   7: XIC(L_PD_IN[0].4)OTE(Motor_Turning);
   8: XIC(L_PD_IN[0].5)OTE(Referenced_Drive);
   9: XIC(L_PD_IN[0].6)OTE(NewRelativePosition_Applied);
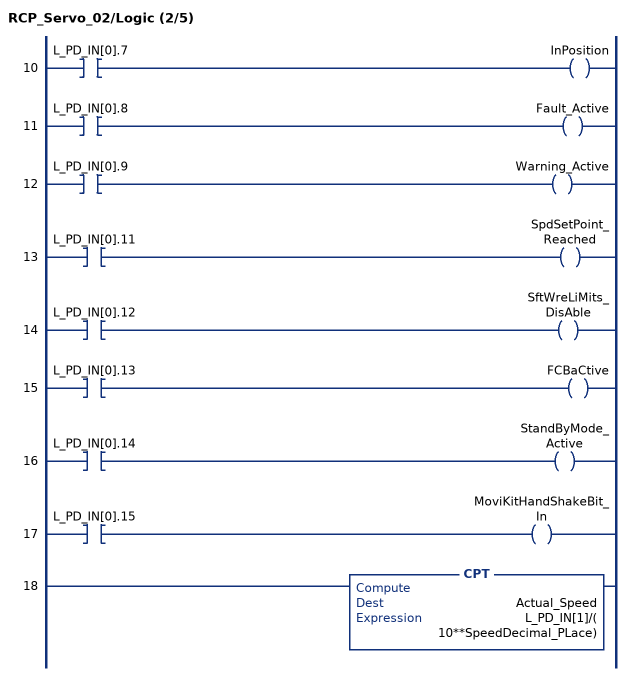
   10: XIC(L_PD_IN[0].7)OTE(InPosition);
   11: XIC(L_PD_IN[0].8)OTE(Fault_Active);
   12: XIC(L_PD_IN[0].9)OTE(Warning_Active);
   13: XIC(L_PD_IN[0].11)OTE(SpdSetPoint_Reached);
   14: XIC(L_PD_IN[0].12)OTE(SftWreLiMits_DisAble);
   15: XIC(L_PD_IN[0].13)OTE(FCBaCtive);
   16: XIC(L_PD_IN[0].14)OTE(StandByMode_Active);
   17: XIC(L_PD_IN[0].15)OTE(MoviKitHandShakeBit_In);
   18: CPT(Actual_Speed,L_PD_IN[1]/(10**SpeedDecimal_PLace));
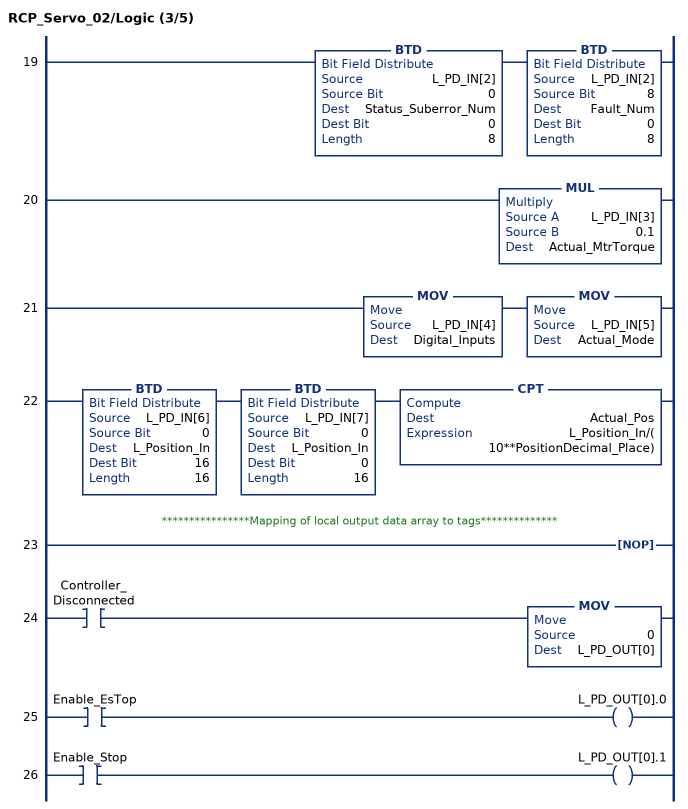
   19: BTD(L_PD_IN[2],0,Status_Suberror_Num,0,8)BTD(L_PD_IN[2],8,Fault_Num,0,8);
   20: MUL(L_PD_IN[3],0.1,Actual_MtrTorque);
   21: MOV(L_PD_IN[4],Digital_Inputs)MOV(L_PD_IN[5],Actual_Mode);
   22: BTD(L_PD_IN[6],0,L_Position_In,16,16)BTD(L_PD_IN[7],0,L_Position_In,0,16)CPT(Actual_Pos,L_Position_In/(10**PositionDecimal_Place));
   // ****************Mapping of local output data array to tags**************
   23: NOP();
   24: XIC(Controller_Disconnected)MOV(0,L_PD_OUT[0]);
   25: XIC(Enable_EsTop)OTE(L_PD_OUT[0].0);
   26: XIC(Enable_Stop)OTE(L_PD_OUT[0].1);
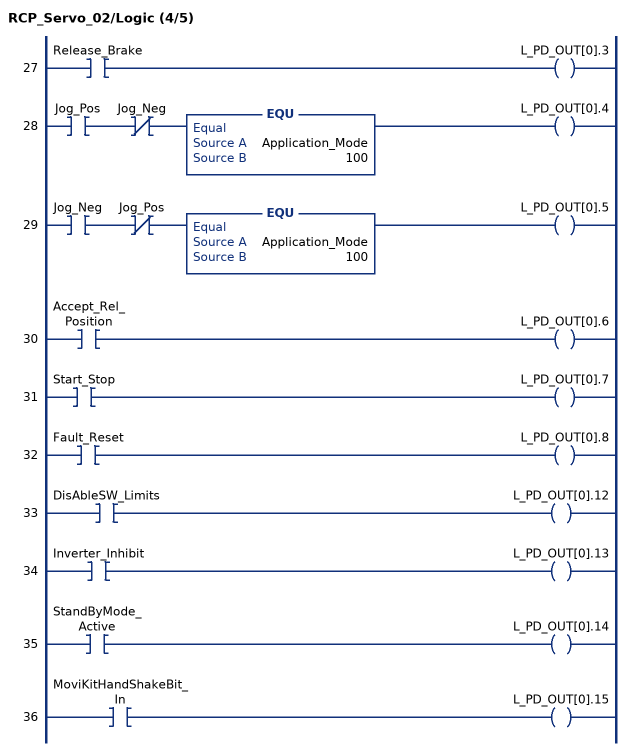
   27: XIC(Release_Brake)OTE(L_PD_OUT[0].3);
   28: XIC(Jog_Pos)XIO(Jog_Neg)EQU(Application_Mode,100)OTE(L_PD_OUT[0].4);
   29: XIC(Jog_Neg)XIO(Jog_Pos)EQU(Application_Mode,100)OTE(L_PD_OUT[0].5);
   30: XIC(Accept_Rel_Position)OTE(L_PD_OUT[0].6);
   31: XIC(Start_Stop)OTE(L_PD_OUT[0].7);
   32: XIC(Fault_Reset)OTE(L_PD_OUT[0].8);
   33: XIC(DisAbleSW_Limits)OTE(L_PD_OUT[0].12);
   34: XIC(Inverter_Inhibit)OTE(L_PD_OUT[0].13);
   35: XIC(StandByMode_Active)OTE(L_PD_OUT[0].14);
   36: XIC(MoviKitHandShakeBit_In)OTE(L_PD_OUT[0].15);
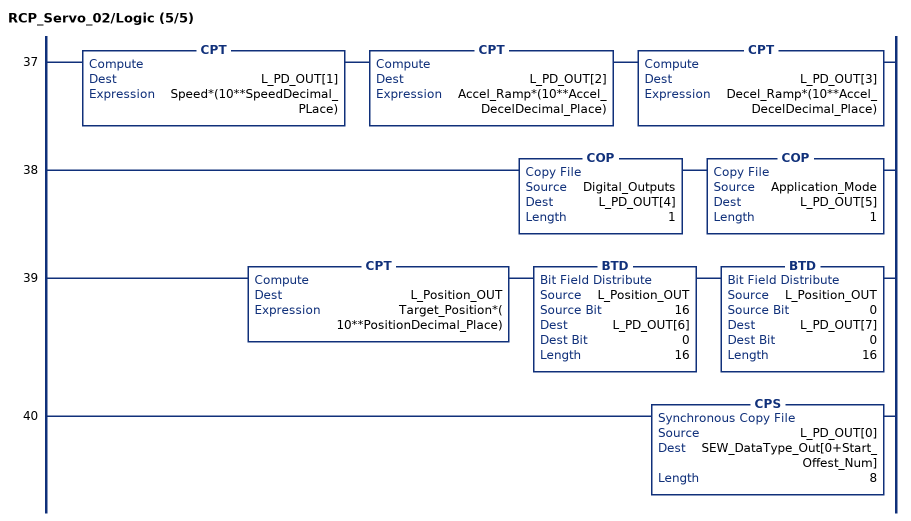
   37: CPT(L_PD_OUT[1],Speed*(10**SpeedDecimal_PLace))CPT(L_PD_OUT[2],Accel_Ramp*(10**Accel_DecelDecimal_Place))CPT(L_PD_OUT[3],Decel_Ramp*(10**Accel_DecelDecimal_Place));
   38: COP(Digital_Outputs,L_PD_OUT[4],1)COP(Application_Mode,L_PD_OUT[5],1);
   39: CPT(L_Position_OUT,Target_Position*(10**PositionDecimal_Place))BTD(L_Position_OUT,16,L_PD_OUT[6],0,16)BTD(L_Position_OUT,0,L_PD_OUT[7],0,16);
   40: CPS(L_PD_OUT[0],SEW_DataType_Out[0+Start_Offest_Num],8);
END_ROUTINE
END_ADD_ON_INSTRUCTION
